# EPICS substitutions: db/Beckhoff_3XXX/ecmcEL3751.substitutions
file "ecmcEcSlave.template"
{
  pattern {}
          {}
}

file "ecmc_analogInput-chX.template"{
  pattern {CH_ID,   EGU,    PREC}
          {01,      "Raw",  3   }
}

file "ecmc_status-chX.template"
{
  pattern {CH_ID, KEY }
          {01,    "AI"}
}
